TYPE Velocityctrl_monitor_typ :
STRUCT
	OrgVelKp        			: LREAL;
	SetCyclicTorque 			: LREAL;
	OrgMaxTorque 				: LREAL;				
	OrgCyclicTorque 			: LREAL;			
	OrgSctrlKp 					: LREAL;
	OrgSctrlKi 					: LREAL;
	OrgGainCtrl 				: LREAL;
	OrgAccToCloseThePosError 	:LREAL; 
END_STRUCT
END_TYPE

(* stored: Version 1.1.0.1, ProductVersion 3.1.4024.3
   DUT Velocityctrl_monitor_typ: Id {b4b72bb1-0dd5-452e-a745-752e9dda2010} *)
